// TwinCAT 3 PLC project IDLoopGW_PLC
// ProgramVersion: 3.1.4024.0
// libraries:
//   Tc2_Standard, * (Beckhoff Automation GmbH)
//   Tc2_System, * (Beckhoff Automation GmbH)
//   Tc3_Module, * (Beckhoff Automation GmbH)
// project tree:
//   DUTs/ HighLow_pointers.TcDUT
//   GVLs/ GVL.TcGVL, Robot_INT_inputs.TcGVL, Robot_INT_outputs.TcGVL
//   / PlcTask.TcTTO
//   POUs/functions/ read_2bytes.TcPOU, write_highbyte.TcPOU, write_lowbyte.TcPOU
//   POUs/ MAIN.TcPOU, Robot_IO_mapping.TcPOU
//   POUs/unused/ int_check.TcPOU, Robot_Input_mapping.TcPOU, Robot_Output_mapping.TcPOU

CONFIGURATION IDLoopGW_PLC
    RESOURCE PLC ON TwinCAT3
        TASK PlcTask(INTERVAL := T#16ms, PRIORITY := 20);
        PROGRAM MAIN WITH PlcTask : MAIN;
    END_RESOURCE
END_CONFIGURATION

// ---- DUTs/HighLow_pointers.TcDUT
TYPE HighLow_pointers :
STRUCT
	pHigh_byte : POINTER TO BYTE;
	pLow_byte : POINTER TO BYTE;
END_STRUCT
END_TYPE

// ---- GVLs/GVL.TcGVL
{attribute 'qualified_only'}
VAR_GLOBAL
	
	G_Dev_state AT%I* : UINT;
	G_Dummy AT%I* :BOOL := FALSE;
	
	
	G_FromYaskawa AT%I* : ARRAY [0..63] OF  BYTE;
	G_ToYaskawa AT%Q* :ARRAY [0..63] OF  BYTE;
	
	
END_VAR

// ---- GVLs/Robot_INT_inputs.TcGVL
{attribute 'qualified_only'}
VAR_GLOBAL
	
	(*_____________Robot Input BOOL parameters__________________*)

	
	
	b_Grundstellung 	: BOOL;
	b_UpdateParam		: BOOL;
	b_Start				: BOOL;
	b_ProgAbbrechen		: BOOL;
	b_Quittieren		: BOOL;	



	(*_____________Robot Input INT parameters__________________*)

	Job_Number :INT;
	Druckskraft :INT;
	Roll_Geschwindigkeit :INT;
	Contact_Angle :INT;
	Frequeny :INT;
	Start_Roll_Angle :INT; 
	End_Roll_Angle :INT;
	FWD_Speed :INT;
	Shift_Speed_X_FWD_Speed :INT;
	Shift_Speed_Y_FWD_Speed :INT;
	Rot_Speed_X :INT;
	Rot_Speed_Y :INT;
	Rot_Speed_Z :INT;
	
	
END_VAR

// ---- GVLs/Robot_INT_outputs.TcGVL
{attribute 'qualified_only'}
VAR_GLOBAL
	
	(*_____________Robot Output BOOL parameters__________________*)
	
	b_IstInGrundstellung 	: BOOL;
	b_Grundstellungen		: BOOL;
	b_ParamGelesen			: BOOL;
	b_Running				: BOOL;
	b_Done					: BOOL;	
	
	(*______________________Error Bits _________________________*)
	Error1					: BOOL;
	Error2					: BOOL;
	Error3					: BOOL;
	Error4					: BOOL;
	Error5					: BOOL;
	Error6					: BOOL;
	Error7					: BOOL;
	Error8					: BOOL;
	Error9					: BOOL;
	Error10					: BOOL;
	Error11					: BOOL;
	Error12					: BOOL;
	Error13					: BOOL;
	Error14					: BOOL;
	Error15					: BOOL;
	Error16					: BOOL;
	
	(*_____________Robot Output INT parameters__________________*)
	
	Job_Number :INT;
	Druckskraft :INT;
	Roll_Geschwindigkeit :INT;
	Contact_Angle :INT;
	Frequeny :INT;
	Start_Roll_Angle :INT; 
	End_Roll_Angle :INT;
	FWD_Speed :INT;
	Shift_Speed_X_FWD_Speed :INT;
	Shift_Speed_Y_FWD_Speed :INT;
	Rot_Speed_X :INT;
	Rot_Speed_Y :INT;
	Rot_Speed_Z :INT;
	
END_VAR

// ---- POUs/MAIN.TcPOU
PROGRAM MAIN
VAR
	dummy :BOOL := FALSE;
END_VAR

//dummy := GVL.G_FromYaskawa[0].1;
//int_check();

Robot_IO_mapping();

END_PROGRAM

// ---- POUs/Robot_IO_mapping.TcPOU
//Map profinet IOs of yasakawa robot to PLC global variables 

PROGRAM Robot_IO_mapping
VAR
	p_jobnumber : POINTER TO BYTE;
END_VAR

(*_____robot's outputs mapping from robot to PLC__________*)

//bool outs
Robot_INT_outputs.b_IstInGrundstellung := GVL.G_FromYaskawa[24].0 ;
Robot_INT_outputs.b_Grundstellungen := GVL.G_FromYaskawa[24].1 ;
Robot_INT_outputs.b_ParamGelesen := GVL.G_FromYaskawa[24].2 ;
Robot_INT_outputs.b_Running := GVL.G_FromYaskawa[24].3 ;
Robot_INT_outputs.b_Done := GVL.G_FromYaskawa[24].4 ;

Robot_INT_outputs.Error1 := GVL.G_FromYaskawa[25].0;
Robot_INT_outputs.Error2 := GVL.G_FromYaskawa[25].1;
Robot_INT_outputs.Error3 := GVL.G_FromYaskawa[25].2;
Robot_INT_outputs.Error4 := GVL.G_FromYaskawa[25].3;
Robot_INT_outputs.Error5 := GVL.G_FromYaskawa[25].4;
Robot_INT_outputs.Error6 := GVL.G_FromYaskawa[25].5;
Robot_INT_outputs.Error7 := GVL.G_FromYaskawa[25].6;
Robot_INT_outputs.Error8 := GVL.G_FromYaskawa[25].7;
Robot_INT_outputs.Error9 := GVL.G_FromYaskawa[26].0;
Robot_INT_outputs.Error10 := GVL.G_FromYaskawa[26].1;
Robot_INT_outputs.Error11 := GVL.G_FromYaskawa[26].2;
Robot_INT_outputs.Error12 := GVL.G_FromYaskawa[26].3;
Robot_INT_outputs.Error13 := GVL.G_FromYaskawa[26].4;
Robot_INT_outputs.Error14 := GVL.G_FromYaskawa[26].5;
Robot_INT_outputs.Error15 := GVL.G_FromYaskawa[26].6;
Robot_INT_outputs.Error16 := GVL.G_FromYaskawa[26].7;

//INT outputs
Robot_INT_outputs.Job_Number := GVL.G_FromYaskawa[27];

Robot_INT_outputs.Druckskraft := read_2bytes(GVL.G_FromYaskawa[29] , GVL.G_FromYaskawa[28]);
Robot_INT_outputs.Roll_Geschwindigkeit := read_2bytes(GVL.G_FromYaskawa[31] , GVL.G_FromYaskawa[30]);
Robot_INT_outputs.Contact_Angle := read_2bytes(GVL.G_FromYaskawa[33] , GVL.G_FromYaskawa[32]);
Robot_INT_outputs.Frequeny := read_2bytes(GVL.G_FromYaskawa[35] , GVL.G_FromYaskawa[34]);
Robot_INT_outputs.Start_Roll_Angle := read_2bytes(GVL.G_FromYaskawa[37] , GVL.G_FromYaskawa[36]);
Robot_INT_outputs.End_Roll_Angle := read_2bytes(GVL.G_FromYaskawa[39] , GVL.G_FromYaskawa[38]);
Robot_INT_outputs.FWD_Speed := read_2bytes(GVL.G_FromYaskawa[41] , GVL.G_FromYaskawa[40]);
Robot_INT_outputs.Shift_Speed_X_FWD_Speed := read_2bytes(GVL.G_FromYaskawa[43] , GVL.G_FromYaskawa[42]);
Robot_INT_outputs.Shift_Speed_Y_FWD_Speed := read_2bytes(GVL.G_FromYaskawa[45] , GVL.G_FromYaskawa[44]);
Robot_INT_outputs.Rot_Speed_X := read_2bytes(GVL.G_FromYaskawa[47] , GVL.G_FromYaskawa[46]);
Robot_INT_outputs.Rot_Speed_Y := read_2bytes(GVL.G_FromYaskawa[49] , GVL.G_FromYaskawa[48]);
Robot_INT_outputs.Rot_Speed_Z := read_2bytes(GVL.G_FromYaskawa[51] , GVL.G_FromYaskawa[50]);



(*_____robot's inputs mapping from plc to robot__________*)

//Bool inputs

Robot_INT_inputs.b_Grundstellung := GVL.G_ToYaskawa[24].0;
Robot_INT_inputs.b_UpdateParam := GVL.G_ToYaskawa[24].1;
Robot_INT_inputs.b_Start := GVL.G_ToYaskawa[24].2;
Robot_INT_inputs.b_ProgAbbrechen := GVL.G_ToYaskawa[24].3;
Robot_INT_inputs.b_Quittieren := GVL.G_ToYaskawa[24].4;

//INT inputs
p_jobnumber := ADR(Robot_INT_inputs.Job_Number);
GVL.G_ToYaskawa[25] := p_jobnumber^; 

GVL.G_ToYaskawa[26] := write_lowbyte(Robot_INT_inputs.Druckskraft); 
GVL.G_ToYaskawa[27] := write_highbyte(Robot_INT_inputs.Druckskraft); 

GVL.G_ToYaskawa[28] := write_lowbyte(Robot_INT_inputs.Roll_Geschwindigkeit); 
GVL.G_ToYaskawa[29] := write_highbyte(Robot_INT_inputs.Roll_Geschwindigkeit); 

GVL.G_ToYaskawa[30] := write_lowbyte(Robot_INT_inputs.Contact_Angle); 
GVL.G_ToYaskawa[31] := write_highbyte(Robot_INT_inputs.Contact_Angle); 

GVL.G_ToYaskawa[32] := write_lowbyte(Robot_INT_inputs.Frequeny); 
GVL.G_ToYaskawa[33] := write_highbyte(Robot_INT_inputs.Frequeny); 

GVL.G_ToYaskawa[34] := write_lowbyte(Robot_INT_inputs.Start_Roll_Angle); 
GVL.G_ToYaskawa[35] := write_highbyte(Robot_INT_inputs.Start_Roll_Angle); 

GVL.G_ToYaskawa[36] := write_lowbyte(Robot_INT_inputs.End_Roll_Angle); 
GVL.G_ToYaskawa[37] := write_highbyte(Robot_INT_inputs.End_Roll_Angle); 

GVL.G_ToYaskawa[38] := write_lowbyte(Robot_INT_inputs.FWD_Speed); 
GVL.G_ToYaskawa[39] := write_highbyte(Robot_INT_inputs.FWD_Speed); 

GVL.G_ToYaskawa[40] := write_lowbyte(Robot_INT_inputs.Shift_Speed_X_FWD_Speed); 
GVL.G_ToYaskawa[41] := write_highbyte(Robot_INT_inputs.Shift_Speed_X_FWD_Speed); 

GVL.G_ToYaskawa[42] := write_lowbyte(Robot_INT_inputs.Shift_Speed_Y_FWD_Speed); 
GVL.G_ToYaskawa[43] := write_highbyte(Robot_INT_inputs.Shift_Speed_Y_FWD_Speed); 

GVL.G_ToYaskawa[44] := write_lowbyte(Robot_INT_inputs.Rot_Speed_X); 
GVL.G_ToYaskawa[45] := write_highbyte(Robot_INT_inputs.Rot_Speed_X); 

GVL.G_ToYaskawa[46] := write_lowbyte(Robot_INT_inputs.Rot_Speed_Y); 
GVL.G_ToYaskawa[47] := write_highbyte(Robot_INT_inputs.Rot_Speed_Y); 

GVL.G_ToYaskawa[48] := write_lowbyte(Robot_INT_inputs.Rot_Speed_Z); 
GVL.G_ToYaskawa[49] := write_highbyte(Robot_INT_inputs.Rot_Speed_Z);

END_PROGRAM

// ---- POUs/functions/read_2bytes.TcPOU
FUNCTION read_2bytes : INT
VAR_INPUT
	gvl_highbyte : BYTE;
	gvl_lowbyte : BYTE;
	
END_VAR
VAR
	//value : INT; 
	p_value : HighLow_pointers; 
END_VAR

p_value.pLow_byte := ADR(read_2bytes);
p_value.pHigh_byte := p_value.pLow_byte +1;
p_value.pLow_byte^ := gvl_lowbyte;
p_value.pHigh_byte^ := gvl_highbyte;

END_FUNCTION

// ---- POUs/functions/write_lowbyte.TcPOU
FUNCTION write_lowbyte : BYTE;

VAR_INPUT
	gvl_in : INT;  // INT var to be written to robots 2 bytes group
	//gvl_highbyte : BYTE; // high byte to be written to robots 2 bytes group
	//gvl_lowbyte : BYTE; // low byte to be written to robots 2 bytes group
END_VAR
VAR
	p_value : HighLow_pointers;
END_VAR

p_value.pLow_byte := ADR(gvl_in);
//p_value.pHigh_byte := p_value.pLow_byte +1; 
//gvl_lowbyte := p_value.pLow_byte^;
write_lowbyte := p_value.pLow_byte^;

END_FUNCTION

// ---- POUs/functions/write_highbyte.TcPOU
FUNCTION write_highbyte : BYTE;

VAR_INPUT
	gvl_in : INT;  // INT var to be written to robots 2 bytes group
	//gvl_highbyte : BYTE; // high byte to be written to robots 2 bytes group
	//gvl_lowbyte : BYTE; // low byte to be written to robots 2 bytes group
END_VAR
VAR
	p_value : HighLow_pointers;
END_VAR

p_value.pLow_byte := ADR(gvl_in);
p_value.pHigh_byte := p_value.pLow_byte +1; 
//gvl_lowbyte := p_value.pLow_byte^;
write_highbyte := p_value.pHigh_byte^;

END_FUNCTION

// ---- POUs/unused/int_check.TcPOU
//for testing only 

PROGRAM int_check
VAR
	Druckskraft 				: HighLow_pointers;
	dummy_in					: HighLow_pointers;
	dummy_val					: INT :=0 ;
	dummy_in_r					: INT ;
	dummy_out_w					: HighLow_pointers ;
	write_test					: write_2bytess;
END_VAR

(*
Druckskraft.pLow_byte := ADR(dummy_val);
Druckskraft.pHigh_byte := Druckskraft.pLow_byte +1; 
GVL.G_ToYaskawa[25] := Druckskraft.pLow_byte^;
GVL.G_ToYaskawa[26] := Druckskraft.pHigh_byte^;
*)

(*
dummy_in.pLow_byte := ADR(dummy_in_r);
dummy_in.pHigh_byte := dummy_in.pLow_byte +1;
dummy_in.pLow_byte^ := GVL.G_FromYaskawa[25];
dummy_in.pHigh_byte^ := GVL.G_FromYaskawa[26];
*)

dummy_in_r := read_2bytes(GVL.G_FromYaskawa[29] , GVL.G_FromYaskawa[28]);
//write_test (gvl_in := Robot_INT_inputs.Druckskraft, gvl_lowbyte := GVL.G_ToYaskawa[25], gvl_highbyte := GVL.G_ToYaskawa[26]);
//dummy_out_w := write_2bytes(Robot_INT_inputs.Druckskraft, GVL.G_ToYaskawa[26], GVL.G_ToYaskawa[25]);
GVL.G_ToYaskawa[26] := write_lowbyte(Robot_INT_inputs.Druckskraft); 
GVL.G_ToYaskawa[27] := write_highbyte(Robot_INT_inputs.Druckskraft);

END_PROGRAM

// ---- POUs/unused/Robot_Input_mapping.TcPOU
//map INT values to Robot

PROGRAM Robot_Input_mapping
VAR
	Druckskraft 				: HighLow_pointers;
	Roll_Geschwindigkeit 		: HighLow_pointers;
	Contact_Angle 				: HighLow_pointers;
	Frequeny 					: HighLow_pointers;
	Start_Roll_Angle 			: HighLow_pointers;
	End_Roll_Angle 				: HighLow_pointers;
	FWD_Speed 					: HighLow_pointers;
	Shift_Speed_X_FWD_Speed 	: HighLow_pointers;
	Shift_Speed_Y_FWD_Speed 	: HighLow_pointers;
	Rot_Speed_X 				: HighLow_pointers;
	Rot_Speed_Y 				: HighLow_pointers;
	Rot_Speed_Z 				: HighLow_pointers;
	

END_VAR


Druckskraft.pLow_byte := ADR(Robot_INT_outputs.Druckskraft);
Druckskraft.pHigh_byte := Druckskraft.pLow_byte +1; 
GVL.G_ToYaskawa[26] := Druckskraft.pLow_byte^;
GVL.G_ToYaskawa[27] := Druckskraft.pHigh_byte^;

Roll_Geschwindigkeit.pLow_byte := ADR(Robot_INT_outputs.Roll_Geschwindigkeit);
Roll_Geschwindigkeit.pHigh_byte := Roll_Geschwindigkeit.pLow_byte +1; 
GVL.G_ToYaskawa[28] := Roll_Geschwindigkeit.pLow_byte^;
GVL.G_ToYaskawa[29] := Roll_Geschwindigkeit.pHigh_byte^;

Contact_Angle.pLow_byte := ADR(Robot_INT_outputs.Contact_Angle);
Contact_Angle.pHigh_byte := Contact_Angle.pLow_byte +1; 
GVL.G_ToYaskawa[30] := Contact_Angle.pLow_byte^;
GVL.G_ToYaskawa[31] := Contact_Angle.pHigh_byte^;

Frequeny.pLow_byte := ADR(Robot_INT_outputs.Frequeny);
Frequeny.pHigh_byte := Frequeny.pLow_byte +1; 
GVL.G_ToYaskawa[32] := Frequeny.pLow_byte^;
GVL.G_ToYaskawa[33] := Frequeny.pHigh_byte^;

Start_Roll_Angle.pLow_byte := ADR(Robot_INT_outputs.Start_Roll_Angle);
Start_Roll_Angle.pHigh_byte := Start_Roll_Angle.pLow_byte +1; 
GVL.G_ToYaskawa[34] := Start_Roll_Angle.pLow_byte^;
GVL.G_ToYaskawa[35] := Start_Roll_Angle.pHigh_byte^;

End_Roll_Angle.pLow_byte := ADR(Robot_INT_outputs.End_Roll_Angle);
End_Roll_Angle.pHigh_byte := End_Roll_Angle.pLow_byte +1; 
GVL.G_ToYaskawa[36] := End_Roll_Angle.pLow_byte^;
GVL.G_ToYaskawa[37] := End_Roll_Angle.pHigh_byte^;

FWD_Speed.pLow_byte := ADR(Robot_INT_outputs.FWD_Speed);
FWD_Speed.pHigh_byte := FWD_Speed.pLow_byte +1; 
GVL.G_ToYaskawa[38] := FWD_Speed.pLow_byte^;
GVL.G_ToYaskawa[39] := FWD_Speed.pHigh_byte^;

Shift_Speed_X_FWD_Speed.pLow_byte := ADR(Robot_INT_outputs.Shift_Speed_X_FWD_Speed);
Shift_Speed_X_FWD_Speed.pHigh_byte := Shift_Speed_X_FWD_Speed.pLow_byte +1; 
GVL.G_ToYaskawa[40] := Shift_Speed_X_FWD_Speed.pLow_byte^;
GVL.G_ToYaskawa[41] := Shift_Speed_X_FWD_Speed.pHigh_byte^;

Shift_Speed_Y_FWD_Speed.pLow_byte := ADR(Robot_INT_outputs.Shift_Speed_Y_FWD_Speed);
Shift_Speed_Y_FWD_Speed.pHigh_byte := Shift_Speed_Y_FWD_Speed.pLow_byte +1; 
GVL.G_ToYaskawa[42] := Shift_Speed_Y_FWD_Speed.pLow_byte^;
GVL.G_ToYaskawa[43] := Shift_Speed_Y_FWD_Speed.pHigh_byte^;

Rot_Speed_X.pLow_byte := ADR(Robot_INT_outputs.Rot_Speed_X);
Rot_Speed_X.pHigh_byte := Rot_Speed_X.pLow_byte +1; 
GVL.G_ToYaskawa[44] := Rot_Speed_X.pLow_byte^;
GVL.G_ToYaskawa[45] := Rot_Speed_X.pHigh_byte^;

Rot_Speed_Y.pLow_byte := ADR(Robot_INT_outputs.Rot_Speed_Y);
Rot_Speed_Y.pHigh_byte := Rot_Speed_Y.pLow_byte +1; 
GVL.G_ToYaskawa[46] := Rot_Speed_Y.pLow_byte^;
GVL.G_ToYaskawa[47] := Rot_Speed_Y.pHigh_byte^;

Rot_Speed_Z.pLow_byte := ADR(Robot_INT_outputs.Rot_Speed_Z);
Rot_Speed_Z.pHigh_byte := Rot_Speed_Z.pLow_byte +1; 
GVL.G_ToYaskawa[48] := Rot_Speed_Z.pLow_byte^;
GVL.G_ToYaskawa[49] := Rot_Speed_Z.pHigh_byte^;

END_PROGRAM

// ---- POUs/unused/Robot_Output_mapping.TcPOU
//map INT values from Robot


PROGRAM Robot_Output_mapping

VAR
	Druckskraft 				: HighLow_pointers;
	Roll_Geschwindigkeit 		: HighLow_pointers;
	Contact_Angle 				: HighLow_pointers;
	Frequeny 					: HighLow_pointers;
	Start_Roll_Angle 			: HighLow_pointers;
	End_Roll_Angle 				: HighLow_pointers;
	FWD_Speed 					: HighLow_pointers;
	Shift_Speed_X_FWD_Speed 	: HighLow_pointers;
	Shift_Speed_Y_FWD_Speed 	: HighLow_pointers;
	Rot_Speed_X 				: HighLow_pointers;
	Rot_Speed_Y 				: HighLow_pointers;
	Rot_Speed_Z 				: HighLow_pointers;
END_VAR

Druckskraft.pLow_byte := ADR(Robot_INT_inputs.Druckskraft);
Druckskraft.pHigh_byte := Druckskraft.pLow_byte +1; 
Druckskraft.pLow_byte^ := GVL.G_FromYaskawa[28];
Druckskraft.pHigh_byte^:= GVL.G_FromYaskawa[29];

Roll_Geschwindigkeit.pLow_byte := ADR(Robot_INT_inputs.Roll_Geschwindigkeit);
Roll_Geschwindigkeit.pHigh_byte := Roll_Geschwindigkeit.pLow_byte +1; 
Roll_Geschwindigkeit.pLow_byte^ := GVL.G_FromYaskawa[30];
Roll_Geschwindigkeit.pHigh_byte^ := GVL.G_FromYaskawa[31];;

Contact_Angle.pLow_byte := ADR(Robot_INT_inputs.Contact_Angle);
Contact_Angle.pHigh_byte := Contact_Angle.pLow_byte +1; 
Contact_Angle.pLow_byte^ := GVL.G_FromYaskawa[32];
Contact_Angle.pHigh_byte^ := GVL.G_FromYaskawa[33];

Frequeny.pLow_byte := ADR(Robot_INT_inputs.Frequeny);
Frequeny.pHigh_byte := Frequeny.pLow_byte +1; 
Frequeny.pLow_byte^ := GVL.G_FromYaskawa[34];
Frequeny.pHigh_byte^ := GVL.G_FromYaskawa[35];

Start_Roll_Angle.pLow_byte := ADR(Robot_INT_inputs.Start_Roll_Angle);
Start_Roll_Angle.pHigh_byte := Start_Roll_Angle.pLow_byte +1; 
Start_Roll_Angle.pLow_byte^ := GVL.G_FromYaskawa[36];
Start_Roll_Angle.pHigh_byte^ := GVL.G_FromYaskawa[37];

End_Roll_Angle.pLow_byte := ADR(Robot_INT_inputs.End_Roll_Angle);
End_Roll_Angle.pHigh_byte := End_Roll_Angle.pLow_byte +1; 
End_Roll_Angle.pLow_byte^ := GVL.G_FromYaskawa[38];
End_Roll_Angle.pHigh_byte^ := GVL.G_FromYaskawa[39];

FWD_Speed.pLow_byte := ADR(Robot_INT_inputs.FWD_Speed);
FWD_Speed.pHigh_byte := FWD_Speed.pLow_byte +1; 
FWD_Speed.pLow_byte^ := GVL.G_FromYaskawa[40];
FWD_Speed.pHigh_byte^ := GVL.G_FromYaskawa[41];

Shift_Speed_X_FWD_Speed.pLow_byte := ADR(Robot_INT_inputs.Shift_Speed_X_FWD_Speed);
Shift_Speed_X_FWD_Speed.pHigh_byte := Shift_Speed_X_FWD_Speed.pLow_byte +1; 
Shift_Speed_X_FWD_Speed.pLow_byte^ := GVL.G_FromYaskawa[42];
Shift_Speed_X_FWD_Speed.pHigh_byte^ := GVL.G_FromYaskawa[43];

Shift_Speed_Y_FWD_Speed.pLow_byte := ADR(Robot_INT_inputs.Shift_Speed_Y_FWD_Speed);
Shift_Speed_Y_FWD_Speed.pHigh_byte := Shift_Speed_Y_FWD_Speed.pLow_byte +1; 
Shift_Speed_Y_FWD_Speed.pLow_byte^ := GVL.G_FromYaskawa[44];
Shift_Speed_Y_FWD_Speed.pHigh_byte^ := GVL.G_FromYaskawa[45];

Rot_Speed_X.pLow_byte := ADR(Robot_INT_inputs.Rot_Speed_X);
Rot_Speed_X.pHigh_byte := Rot_Speed_X.pLow_byte +1; 
Rot_Speed_X.pLow_byte^ := GVL.G_FromYaskawa[46];
Rot_Speed_X.pHigh_byte^ := GVL.G_FromYaskawa[47];

Rot_Speed_Y.pLow_byte := ADR(Robot_INT_inputs.Rot_Speed_Y);
Rot_Speed_Y.pHigh_byte := Rot_Speed_Y.pLow_byte +1; 
Rot_Speed_Y.pLow_byte^ := GVL.G_FromYaskawa[48];
Rot_Speed_Y.pHigh_byte^ := GVL.G_FromYaskawa[49];

Rot_Speed_Z.pLow_byte := ADR(Robot_INT_inputs.Rot_Speed_Z);
Rot_Speed_Z.pHigh_byte := Rot_Speed_Z.pLow_byte +1; 
Rot_Speed_Z.pLow_byte^ := GVL.G_FromYaskawa[50];
Rot_Speed_Z.pHigh_byte^ := GVL.G_FromYaskawa[51];

END_PROGRAM
